// Mitsubishi GX Works2 project: Watchdog   PLC: FX3U/FX3UC

PROGRAM MAIN
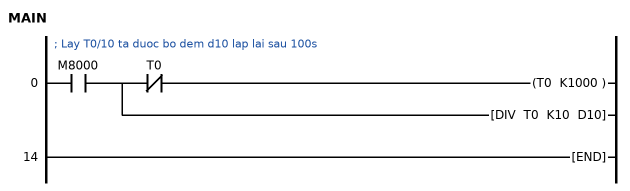
; Lay T0/10 ta duoc bo dem d10 lap lai sau 100s
0     LD      M8000
      MPS
      ANI     T0
      OUT     T0 K1000
      MPP
      DIV     T0 K10 D10
14    END
END_PROGRAM
